// TwinCAT 3 PLC project PLC_HVACBuildingAutomation
// ProgramVersion: 3.1.4026.26
// libraries:
//   Tc2_Standard, * (Beckhoff Automation GmbH)
//   Tc2_System, * (Beckhoff Automation GmbH)
// project tree:
//   DUTs/ FB_AlarmMonitor.TcPOU
//   GVLs/ FB_Damper.TcPOU, FB_Fan.TcPOU
//   / PlcTask.TcTTO
//   POUs/ MAIN.TcPOU
// real-time tasks:
//   TASK PlcTask: cycle T#10ms, priority 20, ADS port 350

CONFIGURATION PLC_HVACBuildingAutomation
    RESOURCE PLC ON TwinCAT3
        TASK PlcTask(INTERVAL := T#10ms, PRIORITY := 20);
        PROGRAM MAIN WITH PlcTask : MAIN;
    END_RESOURCE
END_CONFIGURATION

// ---- POUs/MAIN.TcPOU
PROGRAM MAIN
VAR
	fZoneTemp : REAL := 70.0;  // simulated zone temp, F, starting value
	fSetpoint : REAL := 72.0; // desired temp
	fDeadBand : REAL := 1.0;   // +/- tolerance before acting
	bHeatDemand : BOOL;
	bCoolDemand : BOOL;
	fDriftRate : REAL := 0.02; // simulated passive temp drift per scan
	tSimTimer : TON;
	fbDamper : FB_Damper;
	fbFan : FB_Fan;
	fDamperPosition : REAL;
	fFanSpeed : REAL;
	fbAlarmMonitor : FB_AlarmMonitor;
	bSensorFault : BOOL; // manual test input
	bAckButton : BOOL; // also manual test input
	bHighTempAlarm : BOOL;
	bLowTempAlarm : BOOL;
	bFaultAlarm : BOOL;
	bAnyAlarmActive : BOOL;
END_VAR

// simulated passive temperature drift (zone slowly cools toward 65F baseline)

tSimTimer(IN := TRUE, PT := T#1S);
IF tSimTimer.Q THEN
	IF bHEatDemand THEN
		fZoneTemp := fZoneTemp + 0.5;
	ELSIF bCoolDemand THEN
		fZoneTemp := fZoneTemp - 0.5;
	ELSE
		fZoneTemp := fZoneTemp - fDriftRate; // passive drift toward baseline
	END_IF
	tSimTimer(IN := FALSE);
END_IF

// setpoint / deadband control logic
IF fZoneTemp < (fSetpoint - fDeadband) THEN
	bHeatDemand := TRUE;
	bCoolDemand := FALSE;
ELSIF fZoneTemp > (fSetpoint + fDeadband) THEN
	bCoolDemand := TRUE;
	bHeatDemand := FALSE;
ELSE
	bHeatDemand := FALSE;
	bCoolDemand := FALSE;
END_IF

// Damper and fan control
fbDamper(bCoolDemand := bCoolDemand);
fDamperPosition := fbDamper.fDamperPosition;

fbFan(bHeatDemand := bHeatDemand, bCoolDemand := bCoolDemand);
fFanSpeed := fbFan.fFanSpeed;

// Alarm Monitoring
fbAlarmMonitor(
	fZoneTemp := fZoneTemp,
	bSensorFault := bSensorFault,
	bAckButton := bAckButton
);
bHighTempAlarm := fbAlarmMonitor.bHighTempAlarm;
bLowTempAlarm := fbAlarmMonitor.bLowTempAlarm;
bFaultAlarm := fbAlarmMonitor.bFaultAlarm;
bAnyAlarmActive := fbAlarmMonitor.bAnyAlarmActive;

END_PROGRAM

// ---- GVLs/FB_Damper.TcPOU
FUNCTION_BLOCK FB_Damper
VAR_INPUT
	bCoolDemand : BOOL;
END_VAR
VAR_OUTPUT
	fDamperPosition : REAL; // 0.0 = closed, 100.0 = fully open
END_VAR
VAR
	fRampRate : REAL := 5.0; // % change per scan cycle (simulated actuator speed)
	fTargetPosition : REAL;
END_VAR

// Cooling calls for outside air, damper opens; otherwise closes
IF bCoolDemand THEN
	fTargetPosition := 100.0;
ELSE
	fTargetPosition := 0.0;
END_IF

// Simulate gradual actuator movement
IF fDamperPosition < fTargetPosition THEN
	fDamperPosition := fDamperPosition + fRampRate;
	IF fDamperPosition > fTargetPosition THEN
		fDamperPosition := fTargetPosition;
	END_IF
ELSIF fDamperPosition > fTargetPosition THEN
	fDamperPosition := fDamperPosition - fRampRate;
	IF fDamperPosition < fTargetPosition THEN
		fDamperPosition := fTargetPosition;
	END_IF
END_IF

END_FUNCTION_BLOCK

// ---- GVLs/FB_Fan.TcPOU
FUNCTION_BLOCK FB_Fan
VAR_INPUT
	bHeatDemand : BOOL;
	bCoolDemand : BOOL;
END_VAR
VAR_OUTPUT
	fFanSpeed : REAL; // 0.0 = off, 100.0 = full speed
END_VAR
VAR
	fRampRate : REAL := 10.0;
	fTargetSpeed : REAL;
END_VAR

// Fan runs whenever there's active heating or cooling demand
IF bHeatDemand OR bCoolDemand THEN
	fTargetSpeed := 75.0; // normal operating speed
ELSE
	fTargetSpeed := 0.0;
END_IF

IF fFanSpeed < fTargetSpeed THEN
	fFanSpeed := fFanSpeed + fRampRate;
	IF fFanSpeed > fTargetSpeed THEN
		fFanSpeed := fTargetSpeed;
	END_IF
ELSIF fFanSpeed > fTargetSpeed THEN
	fFanSpeed := fFanSpeed - fRampRate;
	IF fFanSpeed < fTargetSpeed THEN
		fFanSpeed := fTargetSpeed;
	END_IF
END_IF

END_FUNCTION_BLOCK

// ---- DUTs/FB_AlarmMonitor.TcPOU
FUNCTION_BLOCK FB_AlarmMonitor
VAR_INPUT
	fZoneTemp : REAL;
	fHighLimit : REAL := 85.0;
	fLowLimit : REAL := 55.0;
	bSensorFault : BOOL; // simulated fault input
	bAckButton : BOOL; // operator acknowledge/reset
END_VAR
VAR_OUTPUT
	bHighTempAlarm : BOOL;
	bLowTempAlarm : BOOL;
	bFaultAlarm : BOOL;
	bAnyAlarmActive : BOOL;
END_VAR
VAR
	rtrigAck : R_TRIG;
END_VAR

rtrigAck(CLK := bAckButton);

// High temp alarm latches on, clears only on ack one condition is gone
IF fZoneTemp > fHighLimit THEN
	bHighTempAlarm := TRUE;
ELSIF rtrigAck.Q AND fZoneTemp <= fHighLimit THEN
	bHighTempAlarm := FALSE;
END_IF

// Low temp alarm, same pattern
IF fZoneTemp < fLowLimit THEN
	bLowTempAlarm := TRUE;
ELSIF rtrigAck.Q AND fZoneTemp >= fLowLimit THEN
	bLowTempAlarm := FALSE;
END_IF

// Sensor fault alarm, same latch/ack pattern
IF bSensorFault THEN
	bFaultAlarm := TRUE;
ELSIF rtrigAck.Q AND NOT bSensorFault THEN
	bFaultAlarm := FALSE;
END_IF

bAnyAlarmActive := bHighTempAlarm OR bLowTempAlarm OR bFaultAlarm;

END_FUNCTION_BLOCK
